{attribute addProperty BoxType "EP2816-0004-0016"}
{attribute addProperty Id "DO_Outputs_ChannelAT %Q*ARRAY[0..1] OF DO_Outputs_Channel_33B76376128160WcStateAT %I*WcState_64F6A8C6810InfoDataAT %I*InfoData_BC63D37F80100"}
{attribute addProperty CRC "3446843764"}
{attribute addProperty SizeInBites "216"}
{attribute addProperty SizeInBytes "27"}
TYPE EP2816_0ADDCDDB :
STRUCT
	{attribute addProperty Name "DO_Outputs_Channel"}
	DO_Outputs_Channel : ARRAY[0..1] OF DO_Outputs_Channel_33B76376;
	{attribute addProperty Name "WcState"}
	WcState : WcState_64F6A8C6;
	{attribute addProperty Name "InfoData"}
	InfoData : InfoData_BC63D37F;
END_STRUCT
END_TYPE

(* stored: Version 1.2.0.0, ProductVersion 3.1.4024.9
   DUT EP2816_0ADDCDDB: Id {31cbf950-338c-47e0-8745-8d66472273dd} *)
